// Single character string.
TYPE FsT_Char : STRING(1); END_TYPE

(* stored: Version 1.1.0.1, ProductVersion 3.1.4024.4
   DUT FsT_Char: Id {9e593f4d-29d4-4a60-9d59-2066faeae2b1} *)
